(*Vincent Molenkamp : 519540*)
FUNCTION_BLOCK Start_Stop
VAR_INPUT
	START_STOP : BOOL;
	EM_STOP : BOOL;
END_VAR
VAR_OUTPUT
	SystemOn : BOOL;
	State : INT;
END_VAR

VAR
	X: INT;
END_VAR

CASE X OF
	0: IF START_STOP THEN
		SystemOn := 1;
		X := 1;
		END_IF;
	1: IF NOT START_STOP THEN
			X := 2;
		END_IF;
	2: IF START_STOP THEN
		SystemOn := 0;
		END_IF;	
	3: IF NOT START_STOP THEN
		X := 0;	
		END_IF;
	END_CASE
	
	IF NOT EM_STOP THEN
	X := 4;
	SystemOn := 0;
	END_IF; 
	
	IF X = 4 AND EM_STOP AND NOT START_STOP THEN
		X := 0;
	END_IF

END_FUNCTION_BLOCK

(* stored: Version 1.1.0.1, ProductVersion 3.1.4024.12
   POU Start_Stop: Id {687c6edb-2e20-4d80-bd36-dbbef02da369}, SpecialFunc None *)
